SUBAPPLICATION Uebung_172c_ASRT (* Exercise for ASRT_AX_T_FF_SR, ueber AE-Adapter mit logiBUS_IEA statt logiBUS_IE+AE_EVENT_TO_E *)
  (* Standard: 61499-2; Description: Copyright (c) 2026 Meisterschulen am Ostbahnhof This program and the accompanying materials are made available under the terms of the Eclipse Public License 2.0 which is available at https://www.eclipse.org/legal/epl-2.0/ SPDX-License-Identifier: EPL-2.0 *)
  (* Version 1.0, 2026-09-07, Franz Höpfinger, Meisterschulen am Ostbahnhof, initial API and implementation and/or initial documentation *)
  PACKAGE Uebungen;
  IMPORT logiBUS::io::DI::logiBUS_DI::Input_I1;
  IMPORT logiBUS::io::DI::logiBUS_DI::Input_I2;
  IMPORT logiBUS::io::DI::logiBUS_DI::Input_I3;
  IMPORT logiBUS::io::DI::logiBUS_DI_Events::BUTTON_SINGLE_CLICK;
  IMPORT logiBUS::io::DQ::logiBUS_DO::Output_Q1;
  (* Documentation:
  SET/RESET/TOGGLE über AE-Adapter mit logiBUS_IEA (AE bereits eingebaut)
   Dieselbe Funktion wie Uebung_172b_ASRT, aber ohne die manuelle AE_EVENT_TO_E-Brücke pro Kanal: logiBUS_IEA ersetzt logiBUS_IE und liefert den AE-Plug (IN) bereits eingebaut.
   Funktionsbeschreibung
    - logiBUS_IEA kapselt intern einen logiBUS_IE und leitet dessen Klick-Events direkt auf einen eigenen AE-Plug (IN) um - derselbe Mechanismus wie IX → IXA für Pegelsignale, nur für Event-Eingänge.
   - ASRT_3AE_TO_SRT_1 bekommt seine SET_IN/RESET_IN/ TOGGLE_IN jetzt direkt von den drei logiBUS_IEA-Instanzen, ohne Zwischenbaustein.
    Arbeitsauftrag
   Testen Sie identisch zu Uebung_172_ASRT/Uebung_172b_ASRT: I1 klicken → Q1 EIN, I2 klicken → Q1 AUS, I3 klicken → Q1 wechselt den Zustand. Vergleichen Sie alle drei SubApps im Editor: gleiches Verhalten, aber Uebung_172c_ASRT kommt mit den wenigsten Bausteinen aus.
  *)
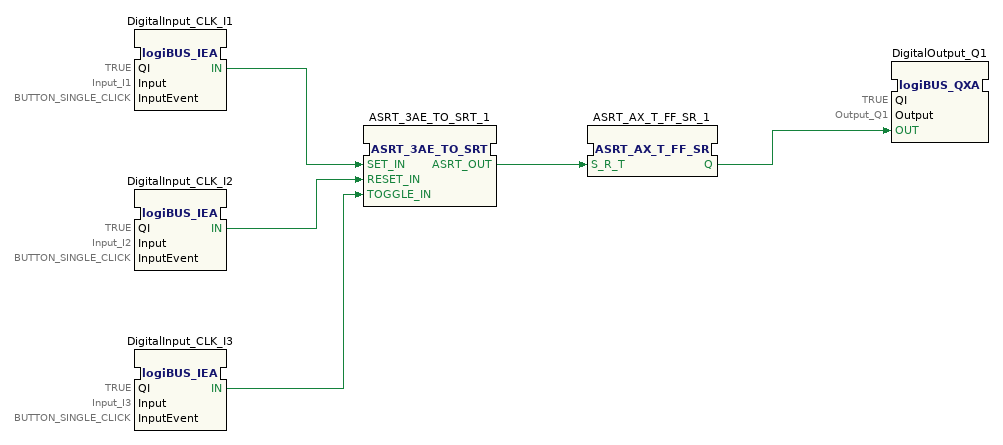
  (* Vergleich zu Uebung_172b_ASRT: dort baute je ein AE_EVENT_TO_E die Bruecke vom rohen logiBUS_IE-Klick-Event zum AE-Plug. Hier liefert logiBUS_IEA (statt logiBUS_IE) den AE-Plug bereits eingebaut - dieselbe Bruecke steckt schon im Baustein, kein separates AE_EVENT_TO_E noetig. *)
  FBS
    ASRT_AX_T_FF_SR_1 : adapter::events::unidirectional::ASRT_AX_T_FF_SR;
    ASRT_3AE_TO_SRT_1 : adapter::conversion::unidirectional::ASRT_3AE_TO_SRT;
    DigitalInput_CLK_I1 : logiBUS::io::DI::logiBUS_IEA(QI := TRUE, Input := Input_I1, InputEvent := BUTTON_SINGLE_CLICK);
    DigitalOutput_Q1 : logiBUS::io::DQ::logiBUS_QXA(QI := TRUE, Output := Output_Q1);
    DigitalInput_CLK_I2 : logiBUS::io::DI::logiBUS_IEA(QI := TRUE, Input := Input_I2, InputEvent := BUTTON_SINGLE_CLICK);
    DigitalInput_CLK_I3 : logiBUS::io::DI::logiBUS_IEA(QI := TRUE, Input := Input_I3, InputEvent := BUTTON_SINGLE_CLICK);
  END_FBS
  ADAPTER_CONNECTIONS
    DigitalInput_CLK_I1.IN TO ASRT_3AE_TO_SRT_1.SET_IN;
    DigitalInput_CLK_I2.IN TO ASRT_3AE_TO_SRT_1.RESET_IN;
    DigitalInput_CLK_I3.IN TO ASRT_3AE_TO_SRT_1.TOGGLE_IN;
    ASRT_3AE_TO_SRT_1.ASRT_OUT TO ASRT_AX_T_FF_SR_1.S_R_T;
    ASRT_AX_T_FF_SR_1.Q TO DigitalOutput_Q1.OUT;
  END_CONNECTIONS
END_SUBAPPLICATION
